// This function has been automatically generated from the project information.
{attribute 'signature_flag' := '1073741824'}
{attribute 'TcGenerated'}
{attribute 'no-analysis'}
FUNCTION F_GetTitle : WSTRING
VAR_INPUT
	
END_VAR

F_GetTitle := "RoboConnect";

END_FUNCTION

(* stored: Version 1.1.0.1
   POU F_GetTitle: Id {457b79f1-3727-4b78-baa3-d32dd7a23927}, SpecialFunc None *)
